Yaskawa INFORM job: profile_short_planes_program.JBI

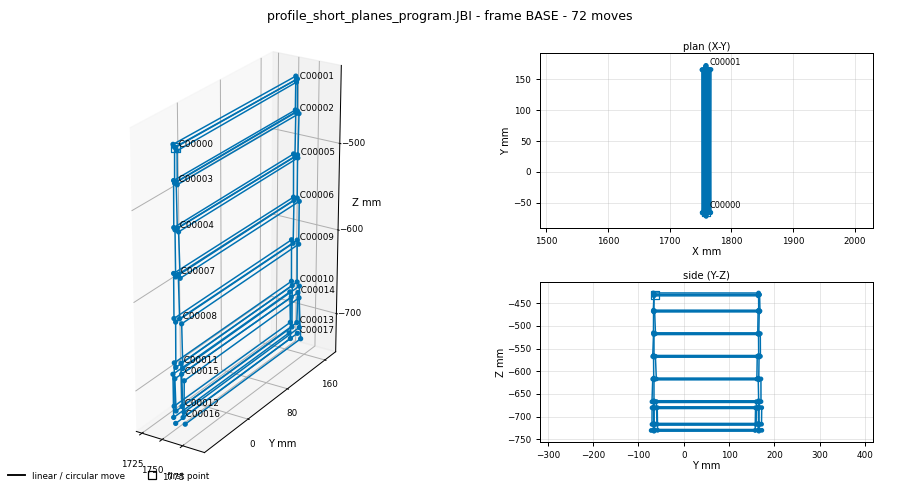
[picture p0: tool path of profile_short_planes_program.JBI in frame BASE, 72 of 77 moves have a stored position in this frame; points joined in program order, loops and branches not executed]
/JOB
//NAME profile_short_planes_program
//POS
///NPOS 72,0,72,0,0,0
///TOOL 0
///POSTYPE BASE
///RECTAN
///RCONF 0,0,0,0,0,0,0,0,0,0,0,0,0,0,0,0,0,0,0,0,0,0,0,0
C00000=1758.200606,-64.385635,-430.952370,5.000000,-89.858167,-175.000000
C00001=1758.182453,167.428392,-430.933415,5.000000,-89.858167,-175.000000
C00002=1758.082575,168.273416,-467.011863,5.000000,-89.858167,-175.000000
C00003=1758.461081,-64.369969,-467.029994,5.000000,-89.858167,-175.000000
C00004=1757.812368,-62.464719,-517.031596,5.000000,-89.858167,-175.000000
C00005=1758.497312,168.984719,-517.010931,5.000000,-89.858167,-175.000000
C00006=1758.542542,169.242210,-567.010951,5.000000,-89.858167,-175.000000
C00007=1758.396503,-62.619338,-567.030317,5.000000,-89.858167,-175.000000
C00008=1757.980592,-60.568676,-617.031331,5.000000,-89.858167,-175.000000
C00009=1758.446685,170.398712,-617.011247,5.000000,-89.858167,-175.000000
C00010=1758.858788,170.540253,-667.010369,5.000000,-89.858167,-175.000000
C00011=1758.893557,-60.445601,-667.029215,5.000000,-89.858167,-175.000000
C00012=1758.774616,-59.241377,-717.029564,5.000000,-89.858167,-175.000000
C00013=1758.432674,171.687215,-717.011483,5.000000,-89.858167,-175.000000
C00014=1759.176930,172.114695,-680.407219,5.000000,-89.858167,-175.000000
C00015=1758.310147,-58.556546,-680.428270,5.000000,-89.858167,-175.000000
C00016=1758.952041,-57.822531,-730.426775,5.000000,-89.858167,-175.000000
C00017=1758.892086,172.359653,-730.408057,180.000000,-60.000000,0.000000
C00018=1757.199682,-67.104837,-427.100173,175.000000,-89.227699,-5.000000
C00019=1757.520047,165.221316,-427.215327,175.000000,-89.227699,-5.000000
C00020=1757.227073,165.473318,-465.236792,175.000000,-89.227699,-5.000000
C00021=1757.019050,-66.699125,-465.123227,175.000000,-89.227699,-5.000000
C00022=1756.639083,-66.917314,-515.122549,175.000000,-89.227699,-5.000000
C00023=1755.882616,165.048072,-515.223014,175.000000,-89.227699,-5.000000
C00024=1756.105303,165.423153,-565.230743,175.000000,-89.227699,-5.000000
C00025=1755.618773,-66.744992,-565.113426,175.000000,-89.227699,-5.000000
C00026=1755.033062,-66.328986,-615.110277,175.000000,-89.227699,-5.000000
C00027=1754.844162,164.369455,-615.217788,175.000000,-89.227699,-5.000000
C00028=1754.713008,165.396830,-665.221058,175.000000,-89.227699,-5.000000
C00029=1754.645755,-66.270019,-665.109632,175.000000,-89.227699,-5.000000
C00030=1753.625154,-66.107742,-715.100500,175.000000,-89.227699,-5.000000
C00031=1753.930560,165.243304,-715.214986,175.000000,-89.227699,-5.000000
C00032=1752.729134,165.553257,-678.600947,175.000000,-89.227699,-5.000000
C00033=1752.928271,-66.401552,-678.492974,175.000000,-89.227699,-5.000000
C00034=1752.714478,-65.848991,-728.494904,175.000000,-89.227699,-5.000000
C00035=1752.472616,165.415361,-728.601971,180.000000,-60.000000,0.000000
C00036=1758.765392,164.246767,-430.445934,5.000000,-89.989370,175.000000
C00037=1758.028381,-65.762245,-430.447490,5.000000,-89.989370,175.000000
C00038=1758.566832,-67.345048,-467.347821,5.000000,-89.989370,175.000000
C00039=1758.586778,164.143713,-467.346388,5.000000,-89.989370,175.000000
C00040=1758.588371,163.345204,-517.346394,5.000000,-89.989370,175.000000
C00041=1757.968577,-66.774555,-517.347929,5.000000,-89.989370,175.000000
C00042=1759.197461,-68.556797,-567.347713,5.000000,-89.989370,175.000000
C00043=1758.643464,162.239970,-567.346391,5.000000,-89.989370,175.000000
C00044=1758.687896,161.400115,-617.346389,5.000000,-89.989370,175.000000
C00045=1758.467548,-68.528333,-617.347849,5.000000,-89.989370,175.000000
C00046=1759.103563,-70.213568,-667.347742,5.000000,-89.989370,175.000000
C00047=1758.807107,160.235008,-667.346375,5.000000,-89.989370,175.000000
C00048=1759.211695,159.869192,-717.346303,5.000000,-89.989370,175.000000
C00049=1758.634683,-70.164782,-717.347830,5.000000,-89.989370,175.000000
C00050=1757.612557,-70.008341,-680.745479,5.000000,-89.989370,175.000000
C00051=1758.693917,158.474298,-680.743868,5.000000,-89.989370,175.000000
C00052=1758.695350,157.678184,-730.743874,5.000000,-89.989370,175.000000
C00053=1759.186804,-71.955131,-730.745200,180.000000,-60.000000,0.000000
C00054=1758.897476,164.329511,-433.423874,5.000000,-88.978379,175.000000
C00055=1760.845903,-65.667846,-433.521527,5.000000,-88.978379,175.000000
C00056=1760.686834,-65.919747,-469.054865,5.000000,-88.978379,175.000000
C00057=1761.075884,166.653663,-468.914046,5.000000,-88.978379,175.000000
C00058=1760.876059,165.598593,-518.926175,5.000000,-88.978379,175.000000
C00059=1761.489443,-65.773190,-519.048425,5.000000,-88.978379,175.000000
C00060=1762.714813,-65.748961,-569.034518,5.000000,-88.978379,175.000000
C00061=1762.870614,166.258122,-568.898184,5.000000,-88.978379,175.000000
C00062=1763.215068,165.586856,-618.900386,5.000000,-88.978379,175.000000
C00063=1763.840791,-65.730144,-619.022385,5.000000,-88.978379,175.000000
C00064=1764.578792,-65.769152,-669.017205,5.000000,-88.978379,175.000000
C00065=1764.347672,166.172248,-668.887809,5.000000,-88.978379,175.000000
C00066=1765.108634,165.799063,-718.882412,5.000000,-88.978379,175.000000
C00067=1765.421388,-65.748320,-719.010125,5.000000,-88.978379,175.000000
C00068=1766.367210,-66.052810,-682.398851,5.000000,-88.978379,175.000000
C00069=1765.036618,164.533140,-682.289842,5.000000,-88.978379,175.000000
C00070=1766.975334,165.881536,-732.262451,5.000000,-88.978379,175.000000
C00071=1766.672623,-65.650412,-732.401131,180.000000,-60.000000,0.000000
///POSTYPE PULSE
///PULSE
EC00000=4096.0
EC00001=4096.0
EC00002=4096.0
EC00003=4096.0
EC00004=4096.0
EC00005=4096.0
EC00006=4096.0
EC00007=4096.0
EC00008=4096.0
EC00009=4096.0
EC00010=4096.0
EC00011=4096.0
EC00012=4096.0
EC00013=4096.0
EC00014=4096.0
EC00015=4096.0
EC00016=4096.0
EC00017=4096.0
EC00018=96256.0
EC00019=96256.0
EC00020=96256.0
EC00021=96256.0
EC00022=96256.0
EC00023=96256.0
EC00024=96256.0
EC00025=96256.0
EC00026=96256.0
EC00027=96256.0
EC00028=96256.0
EC00029=96256.0
EC00030=96256.0
EC00031=96256.0
EC00032=96256.0
EC00033=96256.0
EC00034=96256.0
EC00035=96256.0
EC00036=188416.0
EC00037=188416.0
EC00038=188416.0
EC00039=188416.0
EC00040=188416.0
EC00041=188416.0
EC00042=188416.0
EC00043=188416.0
EC00044=188416.0
EC00045=188416.0
EC00046=188416.0
EC00047=188416.0
EC00048=188416.0
EC00049=188416.0
EC00050=188416.0
EC00051=188416.0
EC00052=188416.0
EC00053=188416.0
EC00054=280576.0
EC00055=280576.0
EC00056=280576.0
EC00057=280576.0
EC00058=280576.0
EC00059=280576.0
EC00060=280576.0
EC00061=280576.0
EC00062=280576.0
EC00063=280576.0
EC00064=280576.0
EC00065=280576.0
EC00066=280576.0
EC00067=280576.0
EC00068=280576.0
EC00069=280576.0
EC00070=280576.0
EC00071=280576.0
//INST
///DATE 2023/08/16 15:31
///ATTR SC,RW,RJ
////FRAME BASE
///GROUP1 RB1,ST1
NOP
MOVJ P009 EX000 VJ=15.00
MOVJ C00000 EC00000 VJ=15.0
CALL JOB:SPYON
MOVL C00001 EC00001 V=150.0
MOVL C00002 EC00002 V=150.0
MOVL C00003 EC00003 V=150.0
MOVL C00004 EC00004 V=150.0
MOVL C00005 EC00005 V=150.0
MOVL C00006 EC00006 V=150.0
MOVL C00007 EC00007 V=150.0
MOVL C00008 EC00008 V=150.0
MOVL C00009 EC00009 V=150.0
MOVL C00010 EC00010 V=150.0
MOVL C00011 EC00011 V=150.0
MOVL C00012 EC00012 V=150.0
MOVL C00013 EC00013 V=150.0
MOVL C00014 EC00014 V=150.0
MOVL C00015 EC00015 V=150.0
MOVL C00016 EC00016 V=150.0
MOVL C00017 EC00017 V=150.0
CALL JOB:SPYOF
MOVJ P009 VJ=15.00
MOVJ C00018 EC00018 VJ=15.0
CALL JOB:SPYON
MOVL C00019 EC00019 V=150.0
MOVL C00020 EC00020 V=150.0
MOVL C00021 EC00021 V=150.0
MOVL C00022 EC00022 V=150.0
MOVL C00023 EC00023 V=150.0
MOVL C00024 EC00024 V=150.0
MOVL C00025 EC00025 V=150.0
MOVL C00026 EC00026 V=150.0
MOVL C00027 EC00027 V=150.0
MOVL C00028 EC00028 V=150.0
MOVL C00029 EC00029 V=150.0
MOVL C00030 EC00030 V=150.0
MOVL C00031 EC00031 V=150.0
MOVL C00032 EC00032 V=150.0
MOVL C00033 EC00033 V=150.0
MOVL C00034 EC00034 V=150.0
MOVL C00035 EC00035 V=150.0
CALL JOB:SPYOF
MOVJ P009 VJ=15.00
MOVJ C00036 EC00036 VJ=15.0
CALL JOB:SPYON
MOVL C00037 EC00037 V=150.0
MOVL C00038 EC00038 V=150.0
MOVL C00039 EC00039 V=150.0
MOVL C00040 EC00040 V=150.0
MOVL C00041 EC00041 V=150.0
MOVL C00042 EC00042 V=150.0
MOVL C00043 EC00043 V=150.0
MOVL C00044 EC00044 V=150.0
MOVL C00045 EC00045 V=150.0
MOVL C00046 EC00046 V=150.0
MOVL C00047 EC00047 V=150.0
MOVL C00048 EC00048 V=150.0
MOVL C00049 EC00049 V=150.0
MOVL C00050 EC00050 V=150.0
MOVL C00051 EC00051 V=150.0
MOVL C00052 EC00052 V=150.0
MOVL C00053 EC00053 V=150.0
CALL JOB:SPYOF
MOVJ P009 VJ=15.00
MOVJ C00054 EC00054 VJ=15.0
CALL JOB:SPYON
MOVL C00055 EC00055 V=150.0
MOVL C00056 EC00056 V=150.0
MOVL C00057 EC00057 V=150.0
MOVL C00058 EC00058 V=150.0
MOVL C00059 EC00059 V=150.0
MOVL C00060 EC00060 V=150.0
MOVL C00061 EC00061 V=150.0
MOVL C00062 EC00062 V=150.0
MOVL C00063 EC00063 V=150.0
MOVL C00064 EC00064 V=150.0
MOVL C00065 EC00065 V=150.0
MOVL C00066 EC00066 V=150.0
MOVL C00067 EC00067 V=150.0
MOVL C00068 EC00068 V=150.0
MOVL C00069 EC00069 V=150.0
MOVL C00070 EC00070 V=150.0
MOVL C00071 EC00071 V=150.0
CALL JOB:SPYOF
MOVJ P009 VJ=15.00
END
